(* Logix 5000 project; controller cal1632 1756-L62 rev 16.20; software revision 16.05 *)

TASK MainTask (continuous, watchdog 500 ms) : P01_System, P02_MOP_HMI_Iface, P11_Zone_1, P12_Zone_2, P13_Zone_3, P19_Advanced_Cooling, P20_Letoff, P21_Splice_Press, P22_Tension_Stand_1

MODULES
   Local : 1756-L62 (ICP 0, rev 16.20)
      p00_di_01 : 1756-IB16 (ICP 4, rev 3.1, Input RPI 20 ms)
      p00_di_02 : 1756-IB16 (ICP 5, rev 3.1, Input RPI 20 ms)
      p00_di_03 : 1756-IB16 (ICP 6, rev 3.1, Input RPI 20 ms)
      p00_do_01 : 1756-OA16I (ICP 7, rev 3.1, Output RPI 20 ms)
      p00_ai_01 : 1756-IF16 (ICP 3, rev 1.1, Input RPI 100 ms)
      Enet_A : 1756-ENBT (Ethernet 10.0.0.1, ICP 1, rev 4.1)
         p00_io_letoff : 1794-AENT (Ethernet 10.0.0.10, rev 3.1, Output RPI 25 ms)
            p00_io_letoff_do_01 : vendor 1 type 7 code 35 (Flex 3, rev 1.1)
            p00_io_letoff_di_01 : 1794-IB16 (Flex 4, rev 1.1)
            p00_io_letoff_di_02 : 1794-IB16 (Flex 5, rev 1.1)
            p00_io_letoff_di_03 : 1794-IB16 (Flex 6, rev 1.1)
            p00_io_letoff_di_04 : 1794-IB16 (Flex 7, rev 1.1)
            p00_io_letoff_ao_01 : 1794-OE4 (Flex 0, rev 2.1, Output RPI 80 ms)
            p00_io_letoff_ai_01 : vendor 1 type 10 code 25 (Flex 1, rev 2.1, Input RPI 80 ms)
            p00_io_letoff_tc_01 : vendor 1 type 10 code 28 (Flex 2, rev 1.1, Input RPI 80 ms)
         p00_io_oven : 1794-AENT (Ethernet 10.0.0.11, rev 3.1, Output RPI 25 ms)
            p00_io_oven_di_01 : 1794-IB16 (Flex 3, rev 1.1)
            p00_io_oven_di_02 : 1794-IB16 (Flex 4, rev 1.1)
            p00_io_oven_di_03 : 1794-IB16 (Flex 5, rev 1.1)
            p00_io_oven_ai_01 : vendor 1 type 10 code 25 (Flex 1, rev 2.1, Input RPI 80 ms)
            p00_io_oven_tc_01 : vendor 1 type 10 code 28 (Flex 2, rev 1.1, Input RPI 80 ms)
            p00_io_oven_ao_01 : 1794-OE4 (Flex 0, rev 2.1, Output RPI 80 ms)
         p00_io_winder : 1794-AENT (Ethernet 10.0.0.12, rev 3.1, Output RPI 25 ms)
            p00_io_winder_di_01 : 1794-IB16 (Flex 5, rev 1.1)
            p00_io_winder_do_01 : vendor 1 type 7 code 35 (Flex 4, rev 1.1)
            p00_io_winder_di_02 : 1794-IB16 (Flex 6, rev 1.1)
            p00_io_winder_ao_02 : 1794-OE4 (Flex 1, rev 2.1, Output RPI 80 ms)
            p00_io_winder_ai_01 : vendor 1 type 10 code 25 (Flex 2, rev 2.1, Input RPI 80 ms)
            p00_io_winder_tc_01 : vendor 1 type 10 code 28 (Flex 3, rev 1.1, Input RPI 80 ms)
            p00_io_winder_ao_01 : 1794-OE4 (Flex 0, rev 2.1, Output RPI 80 ms)
         p00_io_line : 1794-AENT (Ethernet 10.0.0.13, rev 3.1, Output RPI 25 ms)
            p00_io_line_do_01 : vendor 1 type 7 code 35 (Flex 1, rev 1.1)
            p00_io_line_di_01 : 1794-IB16 (Flex 2, rev 1.1)
            p00_io_line_di_02 : 1794-IB16 (Flex 3, rev 1.1)
            p00_io_line_ao_01 : 1794-OE4 (Flex 0, rev 2.1, Output RPI 80 ms)
         p00_io_prc : 1794-AENT (Ethernet 10.0.0.14, rev 3.1, Output RPI 25 ms)
            p00_io_prc_di_01 : 1794-IB16 (Flex 1, rev 1.1)
            p00_io_prc_do_01 : vendor 1 type 7 code 35 (Flex 0, rev 1.1)
         p00_vfd_imp_supply : ETHERNET-MODULE (Ethernet 10.0.0.50, rev 1.1, Output RPI 50 ms)
         p00_vfd_z1_recirc : ETHERNET-MODULE (Ethernet 10.0.0.51, rev 1.1, Output RPI 50 ms)
         p00_vfd_z1_exhaust : ETHERNET-MODULE (Ethernet 10.0.0.52, rev 1.1, Output RPI 50 ms)
         p00_vfd_z2_recirc : ETHERNET-MODULE (Ethernet 10.0.0.53, rev 1.1, Output RPI 50 ms)
         p00_vfd_z2_exhaust : ETHERNET-MODULE (Ethernet 10.0.0.54, rev 1.1, Output RPI 50 ms)
         p00_vfd_z3_exhaust : ETHERNET-MODULE (Ethernet 10.0.0.56, rev 1.1, Output RPI 50 ms)
         p00_vfd_z3_recirc : ETHERNET-MODULE (Ethernet 10.0.0.55, rev 1.1, Output RPI 50 ms)
      Enet_B : 1756-ENBT (ICP 2, Ethernet 10.0.1.1, rev 4.1)
         p00_vfd_loa : ETHERNET-MODULE (Ethernet 10.0.1.10, rev 1.1, Output RPI 10 ms)
         p00_vfd_lob : ETHERNET-MODULE (Ethernet 10.0.1.11, rev 1.1, Output RPI 10 ms)
         p00_vfd_lo_turret : ETHERNET-MODULE (Ethernet 10.0.1.12, rev 1.1, Output RPI 10 ms)
         p00_vfd_ts1 : ETHERNET-MODULE (Ethernet 10.0.1.13, rev 1.1, Output RPI 10 ms)
         p00_vfd_mtr : ETHERNET-MODULE (Ethernet 10.0.1.14, rev 1.1, Output RPI 10 ms)
         p00_srv_mtr_os : ETHERNET-MODULE (Ethernet 10.0.1.15, rev 1.1, Output RPI 10 ms)
         p00_srv_mtr_ds : ETHERNET-MODULE (Ethernet 10.0.1.16, rev 1.1, Output RPI 10 ms)
         p00_vfd_ts2 : ETHERNET-MODULE (Ethernet 10.0.1.17, rev 1.1, Output RPI 10 ms)
         p00_vfd_slitter : ETHERNET-MODULE (Ethernet 10.0.1.18, rev 1.1, Output RPI 10 ms)
         p00_vfd_wdr_turret : ETHERNET-MODULE (Ethernet 10.0.1.19, rev 1.1, Output RPI 10 ms)
         p00_vfd_wda : ETHERNET-MODULE (Ethernet 10.0.1.20, rev 1.1, Output RPI 10 ms)
         p00_vfd_wdb : ETHERNET-MODULE (Ethernet 10.0.1.21, rev 1.1, Output RPI 10 ms)
         p00_vfd_sprng : ETHERNET-MODULE (Ethernet 10.0.1.22, rev 1.1, Output RPI 10 ms)
END_MODULES

TYPE Accumulator :
STRUCT
   OUT_Not_EStop : BOOL;   // E-Stop Not Requested
   OUT_Not_Fast_Stop : BOOL;   // Fast Stop Not Requested
   OUT_Not_Normal_Stop : BOOL;   // Normal Stop Not Requested
   OUT_Request_Line_Slowdown : BOOL;   // Request Line Slowdown
   OUT_Full : BOOL;   // Accumulator is Full
   OUT_Empty : BOOL;   // Accumulator is Empty
   OUT_Alarm : BOOL;   // Alarm Exists
   OUT_Unack_Alarm : BOOL;   // Unacknowledged Alarm Exists
   OUT_Warning : BOOL;   // Warning Exists
   OUT_Unack_Warning : BOOL;   // Unacknowledged Warning Exists
   OUT_control_limit : BOOL;   // Control Limit Position
   OUT_Speed : REAL;   // Output Speed
   OUT_Nip_Close : BOOL;   // Nip Close Request
   IN_Speed : REAL;   // Input Speed
   OUT_Acc_Payout : BOOL;   // Accumulator Payout
   OUT_Close_Nip : BOOL;   // Close Nip
   OUT_Acc_Fill_Request : BOOL;   // Accumulator Fill Request
END_STRUCT
END_TYPE

TYPE acs800_di_normal :
STRUCT
   faulted : BOOL;
   warning : BOOL;
   running_fwd : BOOL;
   running_rev : BOOL;
   ready : BOOL;
   ctrl_from_net : BOOL;
   ref_from_net : BOOL;
   at_reference : BOOL;
END_STRUCT
END_TYPE

TYPE acs800_do_normal :
STRUCT
   forward : BOOL;
   reverse : BOOL;
   fault_reset : BOOL;
   net_control : BOOL;
   net_reference : BOOL;
END_STRUCT
END_TYPE

TYPE hmi_dint :
STRUCT
   hmi : DINT[16];
   global : DINT[16];
   zone_1 : DINT[16];
   zone_2 : DINT[16];
   zone_3 : DINT[16];
   letoff : DINT[16];
   ts1 : DINT[16];
   ts2 : DINT[16];
   upl : DINT[16];
   lpl : DINT[16];
   wdr : DINT[16];
   wdt : DINT[16];
   splice : DINT[16];
   mrc : DINT[16];
   static : DINT[16];
   imp : DINT[16];
   misc : DINT[16];
   edg : DINT[16];
   slt : DINT[16];
   impreg : DINT[16];
   adv_cooling : DINT[16];
   retraction : DINT[16];
END_STRUCT
END_TYPE

TYPE hmi_real :
STRUCT
   hmi : REAL[112];
   global : REAL[112];
   zone_1 : REAL[112];
   zone_2 : REAL[112];
   zone_3 : REAL[112];
   letoff : REAL[112];
   ts1 : REAL[112];
   ts2 : REAL[112];
   upl : REAL[112];
   lpl : REAL[112];
   wdr : REAL[112];
   wdt : REAL[112];
   splice : REAL[112];
   mrc : REAL[112];
   static : REAL[112];
   impreg : REAL[112];
   misc : REAL[112];
   edg : REAL[112];
   slt : REAL[112];
   adv_cooling : REAL[112];
END_STRUCT
END_TYPE

TYPE recipe :
STRUCT
   name : STRING;
   comments : STRING;
   master_line_speed : REAL;
   zone_1 : zone;
   zone_2 : zone;
   zone_3 : zone;
   line_speed_sp : REAL;
   letoff_tension_sp : REAL;
   acc_tension_sp : REAL;
   acc_fill_pressure_sp : REAL;
   acc_counter_pressure_sp : REAL;
   cure_time_sp : REAL;
   platen_temp_sp : REAL;
   impreg_gap_sp : REAL;
   impreg_gap_ds_offset_sp : REAL;
   impreg_gap_os_offset_sp : REAL;
   impreg_supply_speed_sp : REAL;
   impreg_roll_speed_sp : REAL;
   ts1_mode_sp : REAL;
   ts1_tension_sp : REAL;
   ts1_stretch_sp : REAL;
   liner_winder_brake_sp : REAL;
   slitter_speed_sp : REAL;
   adv_cooling_temp_sp : REAL;
   ts2_tension_sp : REAL;
   lower_poly_tension_sp : REAL;
   lower_poly_b_tension_sp : REAL;
   upper_poly_tension_sp : REAL;
   upper_poly_b_tension_sp : REAL;
   winder_tension_sp : REAL;
   winder_mode_sp : REAL;
   winder_torque_sp : REAL;
   tension_deviation_sp : REAL;
END_STRUCT
END_TYPE

TYPE routine :
STRUCT
   comment : DINT;
   oneshot : DINT;
   fault : DINT;
   fault_ack : DINT;
   fault1 : DINT;
   fault1_ack : DINT;
   warning : DINT;
   warning_ack : DINT;
   unack_fault : BOOL;
   unack_warning : BOOL;
   state : DINT;
END_STRUCT
END_TYPE

TYPE servo_di :
STRUCT
   mode_bit_0 : BOOL;
   mode_bit_1 : BOOL;
   homed : BOOL;
   stand_still : BOOL;
   at_target_pos : BOOL;
   command_change : BOOL;
   operator_mode_error : BOOL;
   drive_does_not_follow : BOOL;
   actual_op_mode_bit_0 : BOOL;
   actual_op_mode_bit_1 : BOOL;
   class_3_diagnostic : BOOL;
   class_2_diagnostic : BOOL;
   class_1_diagnostic : BOOL;
   operation_bit_14 : BOOL;
   operation_bit_15 : BOOL;
END_STRUCT
END_TYPE

TYPE servo_do :
STRUCT
   command_value_accept : BOOL;
   fault_reset : BOOL;
   jog_forward : BOOL;
   jog_reverse : BOOL;
   jog_enable : BOOL;
   drive_halt_0_halt : BOOL;
   drive_enable : BOOL;
   ready_for_operation_bit_16 : BOOL;
   ready_for_operation_bit_17 : BOOL;
END_STRUCT
END_TYPE

TYPE Setpoint :   // ******************** DO NOT CHANGE ORDER OF TAGS ******************** ****
STRUCT
   SP : REAL;   // Setpoint
   Lo : REAL;   // Lo
   Hi : REAL;   // Hi
END_STRUCT
END_TYPE

TYPE vfd_data :
STRUCT
   In_OutputFreq : DINT;
   In_RPM : DINT;
   In_OutputCurrent : DINT;
   In_MaximumFreq : DINT;
   In_MotorNPHz : DINT;
   In_MotorNPRPM : DINT;
   In_DriveStatus : DINT;
   Out_CommandedFreq : DINT;
   Out_DriveLogicRslt : DINT;
   Out_CommandedRPM : DINT;
   In_DriveStatus_Ready : BOOL;
   In_DriveStatus_Active : BOOL;
   In_DriveStatus_Faulted : BOOL;
   In_DriveStatus_Net : BOOL;
   In_DriveStatus_AtReference : BOOL;
   Out_DriveLogicRslt_Stop : BOOL;
   Out_DriveLogicRslt_Start : BOOL;
   Out_DriveLogicRslt_ClearFault : BOOL;
   Out_DriveLogicRslt_Forward : BOOL;
   Out_DriveLogicRslt_Reverse : BOOL;
END_STRUCT
END_TYPE

TYPE zone :
STRUCT
   recirc_sp : REAL;
   exhaust_sp : REAL;
   temp_sp : REAL;
END_STRUCT
END_TYPE

ADD_ON_INSTRUCTION ABB_PROTOCOL_VFD   (* revision 1.0 *)
VAR_INPUT
   STATUS_WORD : INT; {required}
END_VAR
VAR_OUTPUT
   CONTROL_WORD : INT; {required}
END_VAR
VAR_INPUT
   DRIVE_NOT_READY_FAULT : BOOL;
END_VAR
VAR_OUTPUT
   OUT_FAULT : BOOL; {visible}
   OUT_ALARM : BOOL; {visible}
   OUT_ENABLED : BOOL; {visible}
END_VAR
VAR_INPUT
   IN_START : BOOL; {required}
   IN_GLOBAL_RESET : BOOL; {required}
   IN_DRIVE_PERMISSIVE : BOOL; {required}
END_VAR
VAR
   run_permissive : BOOL;
   enable_drives : BOOL;
   request_run : BOOL;
   drive_on_request : BOOL;
   seq : routine;
   step_3_timer : TIMER := (PRE := 500);
   fault_timer : TIMER := (PRE := 2000);
END_VAR

ROUTINE Logic   (* ladder *)
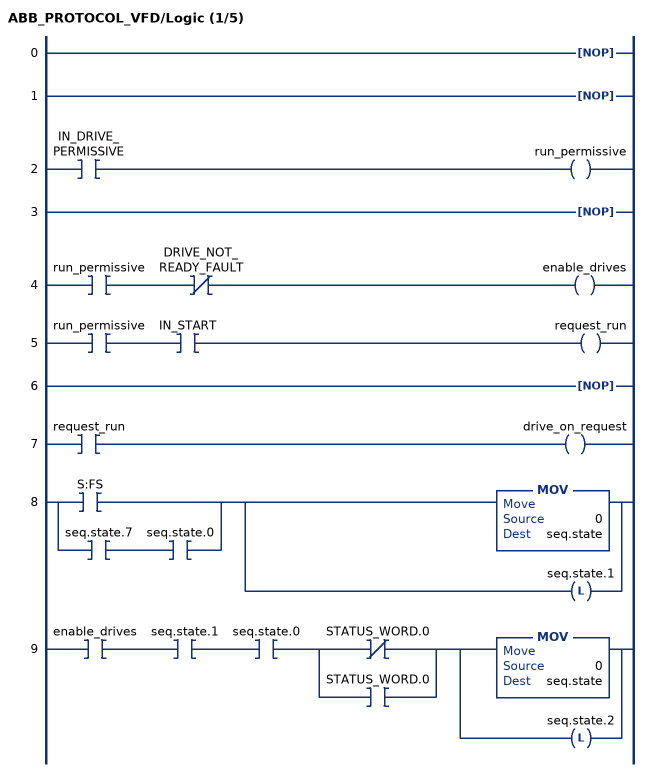
   0: NOP();
   1: NOP();
   2: XIC(IN_DRIVE_PERMISSIVE)OTE(run_permissive);
   3: NOP();
   4: XIC(run_permissive)XIO(DRIVE_NOT_READY_FAULT)OTE(enable_drives);
   5: XIC(run_permissive)XIC(IN_START)OTE(request_run);
   6: NOP();
   7: XIC(request_run)OTE(drive_on_request);
   8: [XIC(S:FS) ,XIC(seq.state.7) XIC(seq.state.0) ][MOV(0,seq.state) ,OTL(seq.state.1) ];
   9: XIC(enable_drives)XIC(seq.state.1)XIC(seq.state.0)[XIO(STATUS_WORD.0) ,XIC(STATUS_WORD.0) ][MOV(0,seq.state) ,OTL(seq.state.2) ];
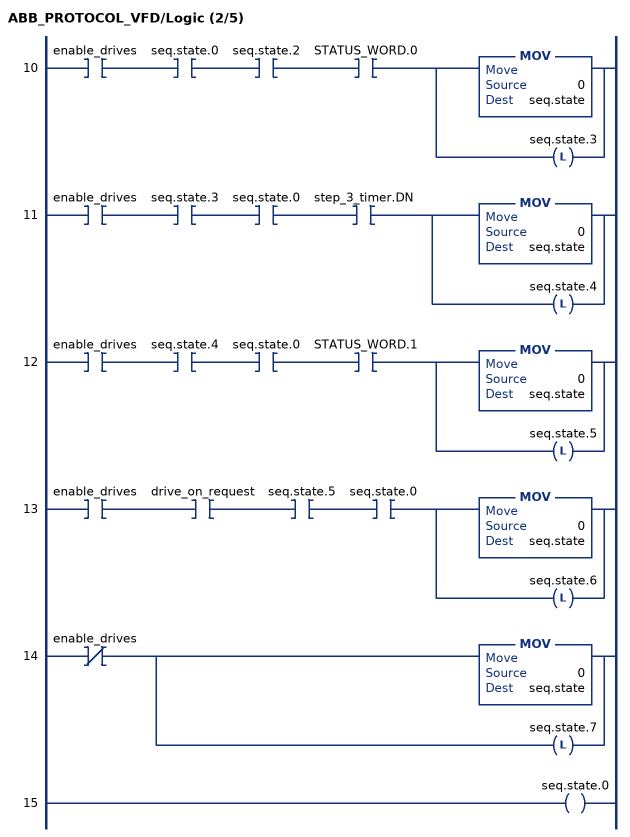
   10: XIC(enable_drives)XIC(seq.state.0)XIC(seq.state.2)XIC(STATUS_WORD.0)[MOV(0,seq.state) ,OTL(seq.state.3) ];
   11: XIC(enable_drives)XIC(seq.state.3)XIC(seq.state.0)XIC(step_3_timer.DN)[MOV(0,seq.state) ,OTL(seq.state.4) ];
   12: XIC(enable_drives)XIC(seq.state.4)XIC(seq.state.0)XIC(STATUS_WORD.1)[MOV(0,seq.state) ,OTL(seq.state.5) ];
   13: XIC(enable_drives)XIC(drive_on_request)XIC(seq.state.5)XIC(seq.state.0)[MOV(0,seq.state) ,OTL(seq.state.6) ];
   14: XIO(enable_drives)[MOV(0,seq.state) ,OTL(seq.state.7) ];
   15: OTE(seq.state.0);
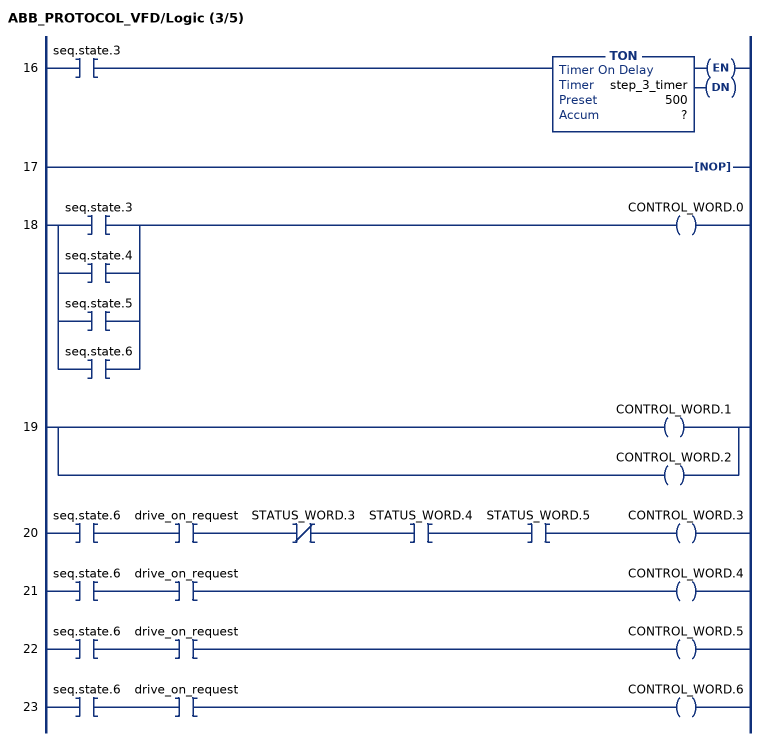
   16: XIC(seq.state.3)TON(step_3_timer,?,?);
   17: NOP();
   18: [XIC(seq.state.3) ,XIC(seq.state.4) ,XIC(seq.state.5) ,XIC(seq.state.6) ]OTE(CONTROL_WORD.0);
   19: [OTE(CONTROL_WORD.1) ,OTE(CONTROL_WORD.2) ];
   20: XIC(seq.state.6)XIC(drive_on_request)XIO(STATUS_WORD.3)XIC(STATUS_WORD.4)XIC(STATUS_WORD.5)OTE(CONTROL_WORD.3);
   21: XIC(seq.state.6)XIC(drive_on_request)OTE(CONTROL_WORD.4);
   22: XIC(seq.state.6)XIC(drive_on_request)OTE(CONTROL_WORD.5);
   23: XIC(seq.state.6)XIC(drive_on_request)OTE(CONTROL_WORD.6);
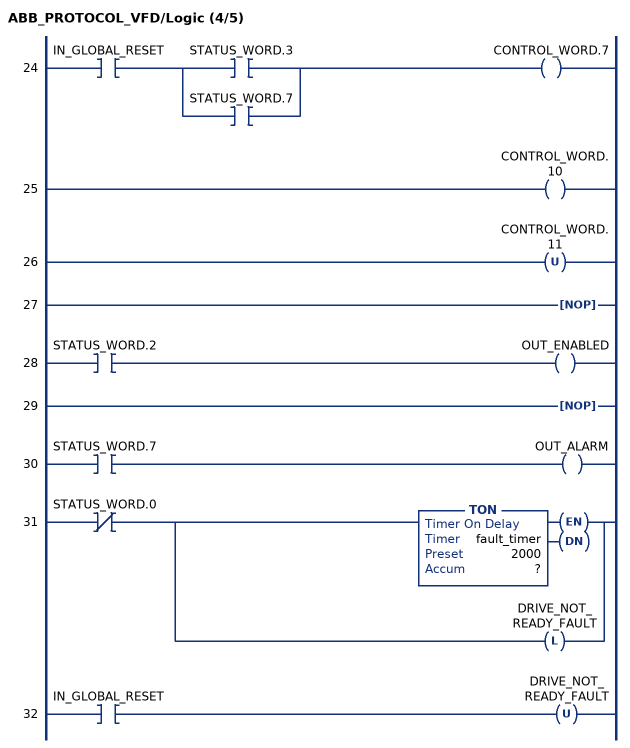
   24: XIC(IN_GLOBAL_RESET)[XIC(STATUS_WORD.3) ,XIC(STATUS_WORD.7) ]OTE(CONTROL_WORD.7);
   25: OTE(CONTROL_WORD.10);
   26: OTU(CONTROL_WORD.11);
   27: NOP();
   28: XIC(STATUS_WORD.2)OTE(OUT_ENABLED);
   29: NOP();
   30: XIC(STATUS_WORD.7)OTE(OUT_ALARM);
   31: XIO(STATUS_WORD.0)[TON(fault_timer,?,?) ,OTL(DRIVE_NOT_READY_FAULT) ];
   32: XIC(IN_GLOBAL_RESET)OTU(DRIVE_NOT_READY_FAULT);
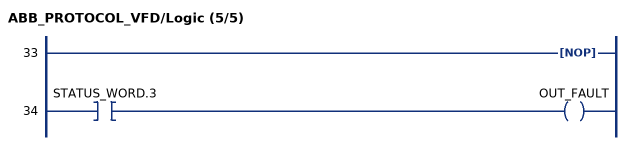
   33: NOP();
   34: XIC(STATUS_WORD.3)OTE(OUT_FAULT);
END_ROUTINE
END_ADD_ON_INSTRUCTION

ADD_ON_INSTRUCTION ARM_PID   (* revision 1.0 *)
VAR_IN_OUT
   PID : PID; {required}
END_VAR
VAR_INPUT
   NOBC : BOOL; {required}
   CA : BOOL; {required}
   Min : REAL; {required}
   Max : REAL; {required}
END_VAR

ROUTINE Logic   (* ladder *)
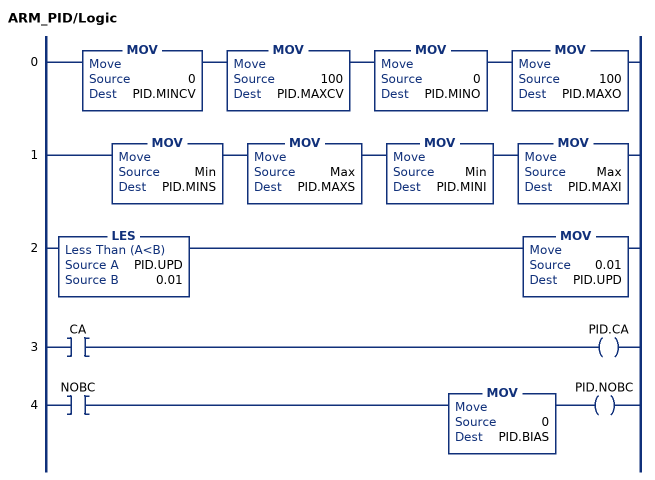
   0: MOV(0,PID.MINCV)MOV(100,PID.MAXCV)MOV(0,PID.MINO)MOV(100,PID.MAXO);
   1: MOV(Min,PID.MINS)MOV(Max,PID.MAXS)MOV(Min,PID.MINI)MOV(Max,PID.MAXI);
   2: LES(PID.UPD,0.01)MOV(0.01,PID.UPD);
   3: XIC(CA)OTE(PID.CA);
   4: XIC(NOBC)MOV(0,PID.BIAS)OTE(PID.NOBC);
END_ROUTINE
END_ADD_ON_INSTRUCTION

ADD_ON_INSTRUCTION Limit_Clamp   (* revision 1.0 *)
VAR_INPUT
   max : REAL; {required}
END_VAR
VAR_IN_OUT
   variable : REAL; {required}
END_VAR
VAR_INPUT
   min : REAL; {required}
END_VAR

ROUTINE Logic   (* ladder *)
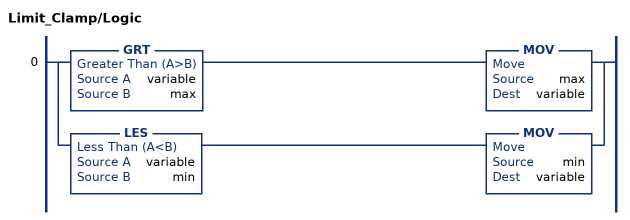
   0: [GRT(variable,max) MOV(max,variable) ,LES(variable,min) MOV(min,variable) ];
END_ROUTINE
END_ADD_ON_INSTRUCTION

ADD_ON_INSTRUCTION Ramp_Test   (* revision 1.0 *)
VAR_INPUT
   SP : REAL; {required}
   Rate : REAL; {required}
   ScanTime : REAL; {required}
END_VAR
VAR_IN_OUT
   PV : REAL; {required}
END_VAR
VAR
   request_decel : BOOL;
   request_accel : BOOL;
END_VAR

ROUTINE Logic   (* ladder *)
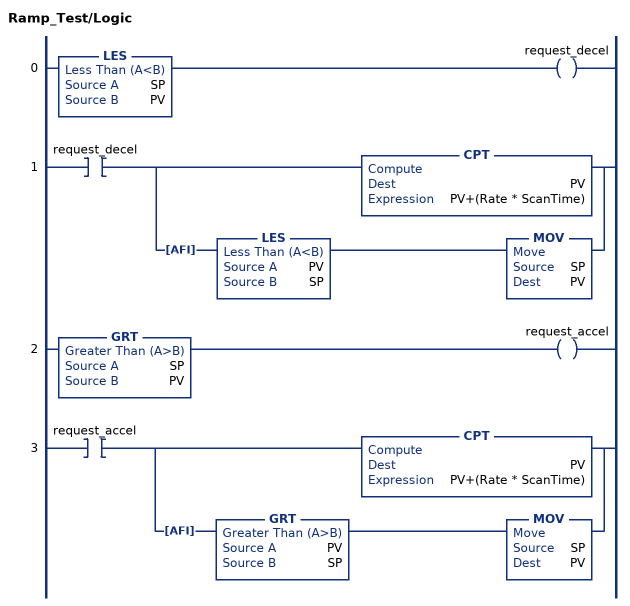
   0: LES(SP,PV)OTE(request_decel);
   1: XIC(request_decel)[CPT(PV,PV+(Rate * ScanTime)) ,AFI() LES(PV,SP) MOV(SP,PV) ];
   2: GRT(SP,PV)OTE(request_accel);
   3: XIC(request_accel)[CPT(PV,PV+(Rate * ScanTime)) ,AFI() GRT(PV,SP) MOV(SP,PV) ];
END_ROUTINE
END_ADD_ON_INSTRUCTION

ADD_ON_INSTRUCTION SYS_ACC_DEC_RAMP   (* revision 1.0 *)
VAR_INPUT
   IN_selected_line_speed : REAL; {required}
   IN_param_master_accel_rate : REAL; {required}
   IN_param_master_decel_rate : REAL; {required}
   IN_last_scan_s : REAL; {required}
END_VAR
VAR_IN_OUT
   IN_OUT_master_ramped_speed : REAL; {required}
END_VAR
VAR
   p01r03_last_scan_ms : DINT;
   local_last_scan_ms : DINT;
END_VAR

ROUTINE Logic   (* ladder *)
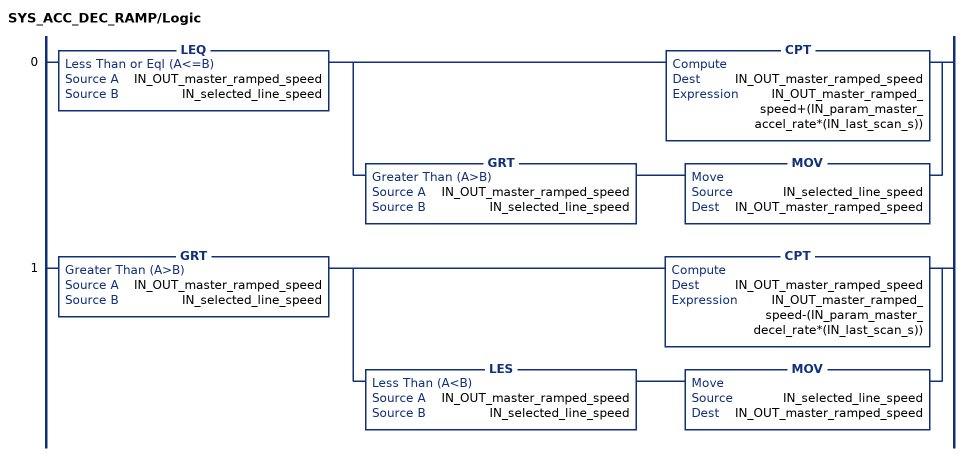
   0: LEQ(IN_OUT_master_ramped_speed,IN_selected_line_speed)[CPT(IN_OUT_master_ramped_speed,IN_OUT_master_ramped_speed+(IN_param_master_accel_rate*(IN_last_scan_s))) ,GRT(IN_OUT_master_ramped_speed,IN_selected_line_speed) MOV(IN_selected_line_speed,IN_OUT_master_ramped_speed) ];
   1: GRT(IN_OUT_master_ramped_speed,IN_selected_line_speed)[CPT(IN_OUT_master_ramped_speed,IN_OUT_master_ramped_speed-(IN_param_master_decel_rate*(IN_last_scan_s))) ,LES(IN_OUT_master_ramped_speed,IN_selected_line_speed) MOV(IN_selected_line_speed,IN_OUT_master_ramped_speed) ];
END_ROUTINE
END_ADD_ON_INSTRUCTION

ADD_ON_INSTRUCTION sys_Acknowledge   (* revision 1.0 *)
VAR_INPUT
   EnableIn1 : BOOL;   // Enable Input - System Defined Parameter
END_VAR
VAR_OUTPUT
   EnableOut1 : BOOL;   // Enable Output - System Defined Parameter
END_VAR
VAR_IN_OUT
   Ack : DINT; {required}
END_VAR
VAR_INPUT
   Alarm : DINT; {required}
END_VAR

ROUTINE Logic   (* ladder *)
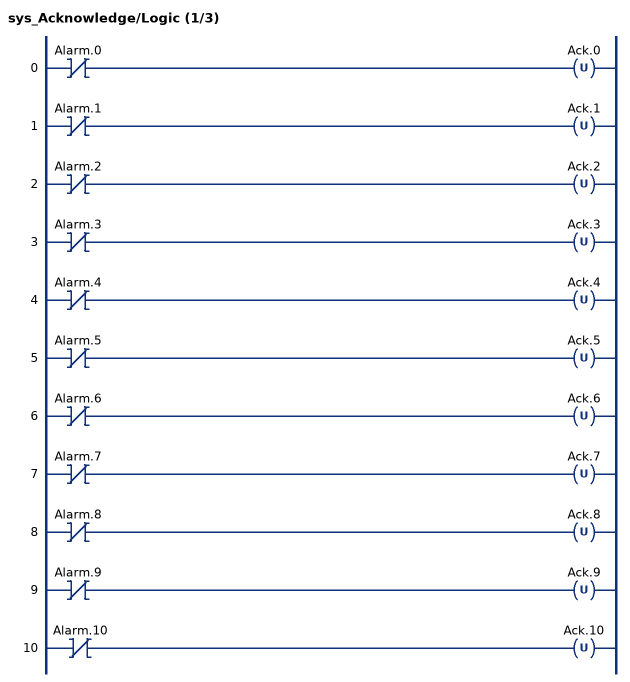
   0: XIO(Alarm.0)OTU(Ack.0);
   1: XIO(Alarm.1)OTU(Ack.1);
   2: XIO(Alarm.2)OTU(Ack.2);
   3: XIO(Alarm.3)OTU(Ack.3);
   4: XIO(Alarm.4)OTU(Ack.4);
   5: XIO(Alarm.5)OTU(Ack.5);
   6: XIO(Alarm.6)OTU(Ack.6);
   7: XIO(Alarm.7)OTU(Ack.7);
   8: XIO(Alarm.8)OTU(Ack.8);
   9: XIO(Alarm.9)OTU(Ack.9);
   10: XIO(Alarm.10)OTU(Ack.10);
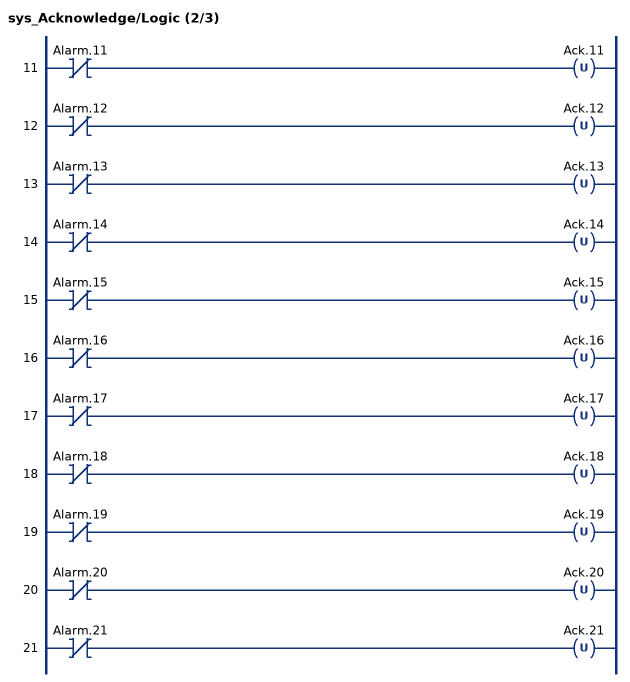
   11: XIO(Alarm.11)OTU(Ack.11);
   12: XIO(Alarm.12)OTU(Ack.12);
   13: XIO(Alarm.13)OTU(Ack.13);
   14: XIO(Alarm.14)OTU(Ack.14);
   15: XIO(Alarm.15)OTU(Ack.15);
   16: XIO(Alarm.16)OTU(Ack.16);
   17: XIO(Alarm.17)OTU(Ack.17);
   18: XIO(Alarm.18)OTU(Ack.18);
   19: XIO(Alarm.19)OTU(Ack.19);
   20: XIO(Alarm.20)OTU(Ack.20);
   21: XIO(Alarm.21)OTU(Ack.21);
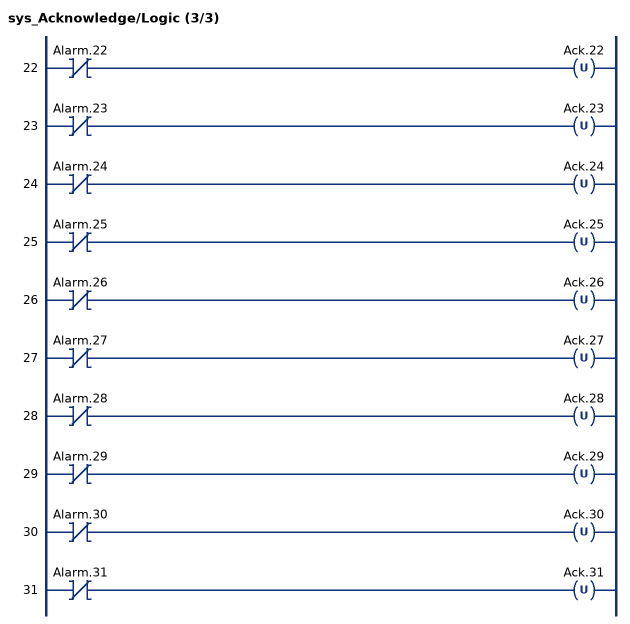
   22: XIO(Alarm.22)OTU(Ack.22);
   23: XIO(Alarm.23)OTU(Ack.23);
   24: XIO(Alarm.24)OTU(Ack.24);
   25: XIO(Alarm.25)OTU(Ack.25);
   26: XIO(Alarm.26)OTU(Ack.26);
   27: XIO(Alarm.27)OTU(Ack.27);
   28: XIO(Alarm.28)OTU(Ack.28);
   29: XIO(Alarm.29)OTU(Ack.29);
   30: XIO(Alarm.30)OTU(Ack.30);
   31: XIO(Alarm.31)OTU(Ack.31);
END_ROUTINE
END_ADD_ON_INSTRUCTION

ADD_ON_INSTRUCTION SYS_ENC   (* revision 1.0 *)
VAR_INPUT
   IN_State : DINT; {required}
END_VAR
VAR_OUTPUT
   OUT_Status : DINT; {required}
END_VAR

ROUTINE Logic   (* ladder *)
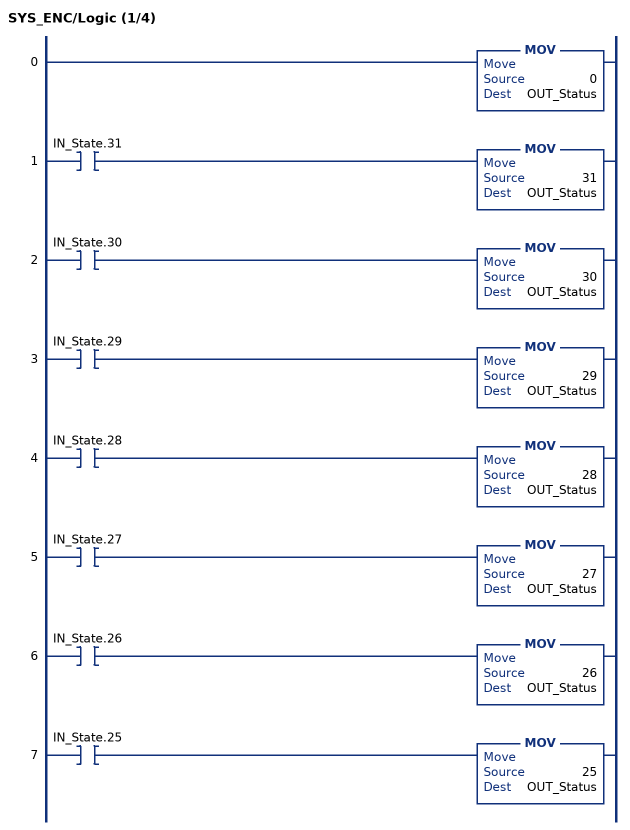
   0: MOV(0,OUT_Status);
   1: XIC(IN_State.31)MOV(31,OUT_Status);
   2: XIC(IN_State.30)MOV(30,OUT_Status);
   3: XIC(IN_State.29)MOV(29,OUT_Status);
   4: XIC(IN_State.28)MOV(28,OUT_Status);
   5: XIC(IN_State.27)MOV(27,OUT_Status);
   6: XIC(IN_State.26)MOV(26,OUT_Status);
   7: XIC(IN_State.25)MOV(25,OUT_Status);
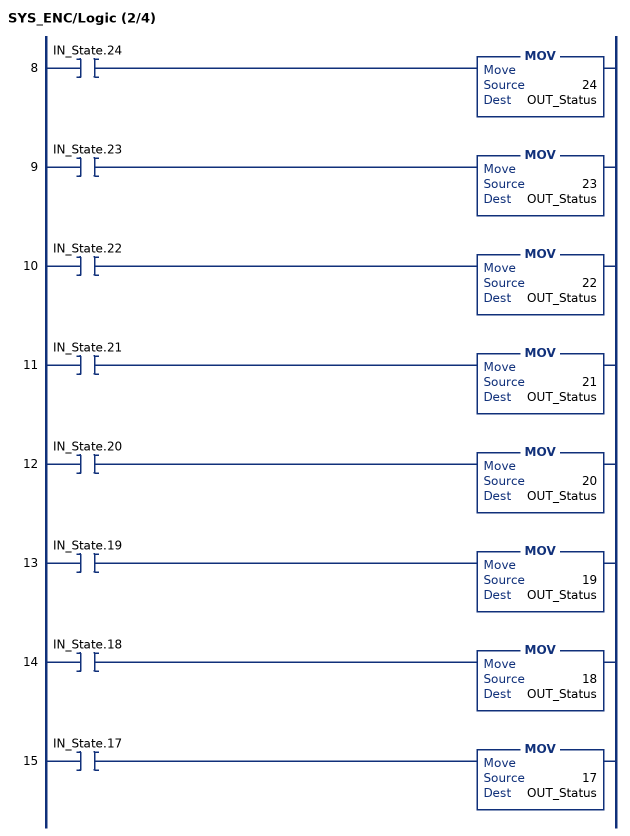
   8: XIC(IN_State.24)MOV(24,OUT_Status);
   9: XIC(IN_State.23)MOV(23,OUT_Status);
   10: XIC(IN_State.22)MOV(22,OUT_Status);
   11: XIC(IN_State.21)MOV(21,OUT_Status);
   12: XIC(IN_State.20)MOV(20,OUT_Status);
   13: XIC(IN_State.19)MOV(19,OUT_Status);
   14: XIC(IN_State.18)MOV(18,OUT_Status);
   15: XIC(IN_State.17)MOV(17,OUT_Status);
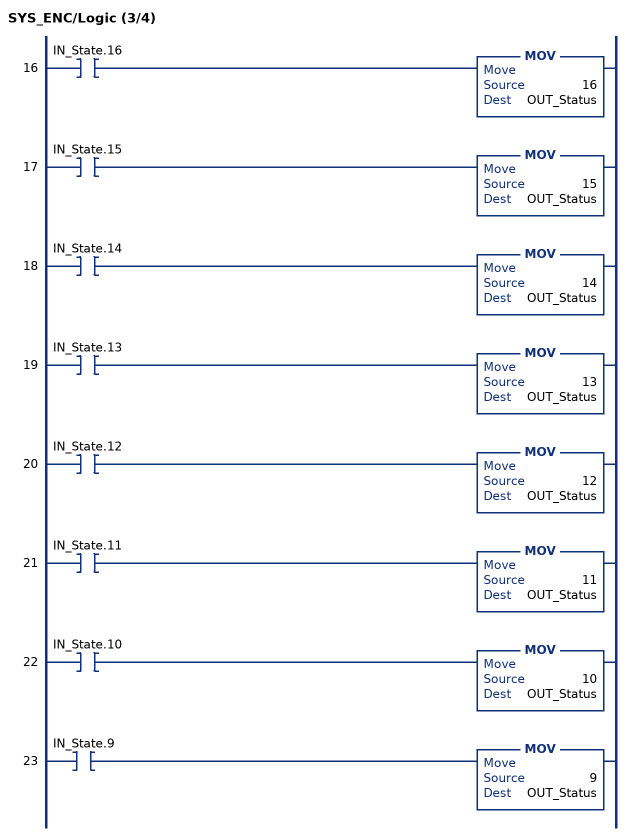
   16: XIC(IN_State.16)MOV(16,OUT_Status);
   17: XIC(IN_State.15)MOV(15,OUT_Status);
   18: XIC(IN_State.14)MOV(14,OUT_Status);
   19: XIC(IN_State.13)MOV(13,OUT_Status);
   20: XIC(IN_State.12)MOV(12,OUT_Status);
   21: XIC(IN_State.11)MOV(11,OUT_Status);
   22: XIC(IN_State.10)MOV(10,OUT_Status);
   23: XIC(IN_State.9)MOV(9,OUT_Status);
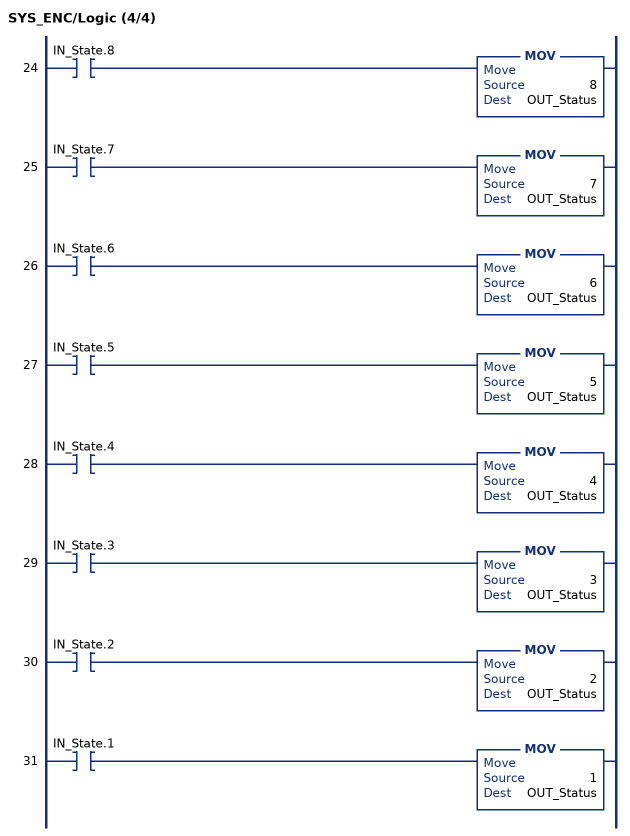
   24: XIC(IN_State.8)MOV(8,OUT_Status);
   25: XIC(IN_State.7)MOV(7,OUT_Status);
   26: XIC(IN_State.6)MOV(6,OUT_Status);
   27: XIC(IN_State.5)MOV(5,OUT_Status);
   28: XIC(IN_State.4)MOV(4,OUT_Status);
   29: XIC(IN_State.3)MOV(3,OUT_Status);
   30: XIC(IN_State.2)MOV(2,OUT_Status);
   31: XIC(IN_State.1)MOV(1,OUT_Status);
END_ROUTINE
END_ADD_ON_INSTRUCTION

ADD_ON_INSTRUCTION SYS_ENC_WITH_ZERO_BIT   (* revision 1.0 *)
VAR_INPUT
   IN_State : DINT; {required}
END_VAR
VAR_OUTPUT
   OUT_Status : DINT; {required}
END_VAR

ROUTINE Logic   (* ladder *)
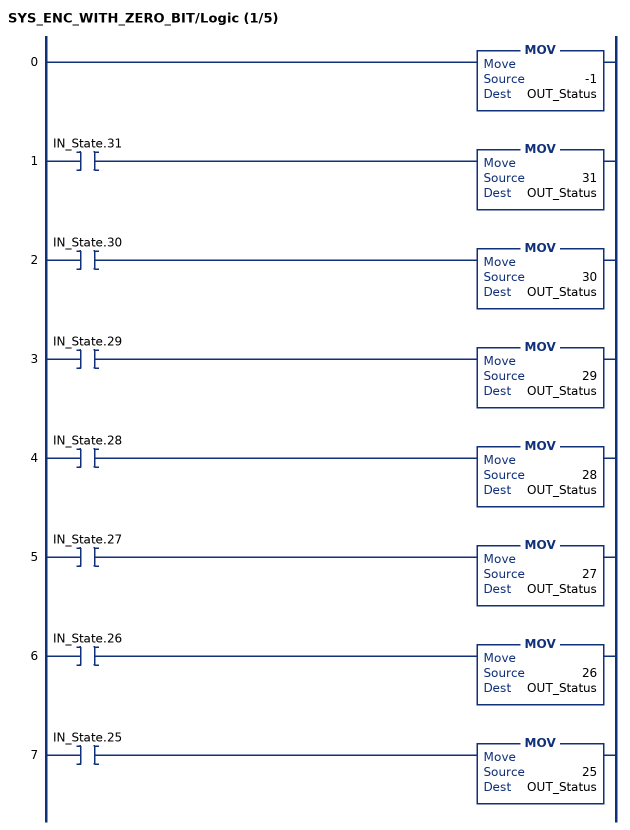
   0: MOV(-1,OUT_Status);
   1: XIC(IN_State.31)MOV(31,OUT_Status);
   2: XIC(IN_State.30)MOV(30,OUT_Status);
   3: XIC(IN_State.29)MOV(29,OUT_Status);
   4: XIC(IN_State.28)MOV(28,OUT_Status);
   5: XIC(IN_State.27)MOV(27,OUT_Status);
   6: XIC(IN_State.26)MOV(26,OUT_Status);
   7: XIC(IN_State.25)MOV(25,OUT_Status);
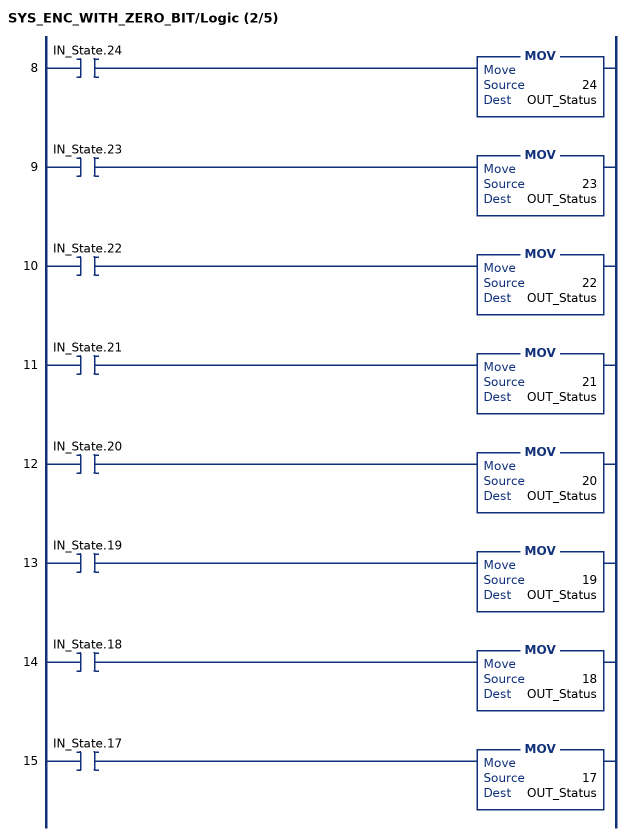
   8: XIC(IN_State.24)MOV(24,OUT_Status);
   9: XIC(IN_State.23)MOV(23,OUT_Status);
   10: XIC(IN_State.22)MOV(22,OUT_Status);
   11: XIC(IN_State.21)MOV(21,OUT_Status);
   12: XIC(IN_State.20)MOV(20,OUT_Status);
   13: XIC(IN_State.19)MOV(19,OUT_Status);
   14: XIC(IN_State.18)MOV(18,OUT_Status);
   15: XIC(IN_State.17)MOV(17,OUT_Status);
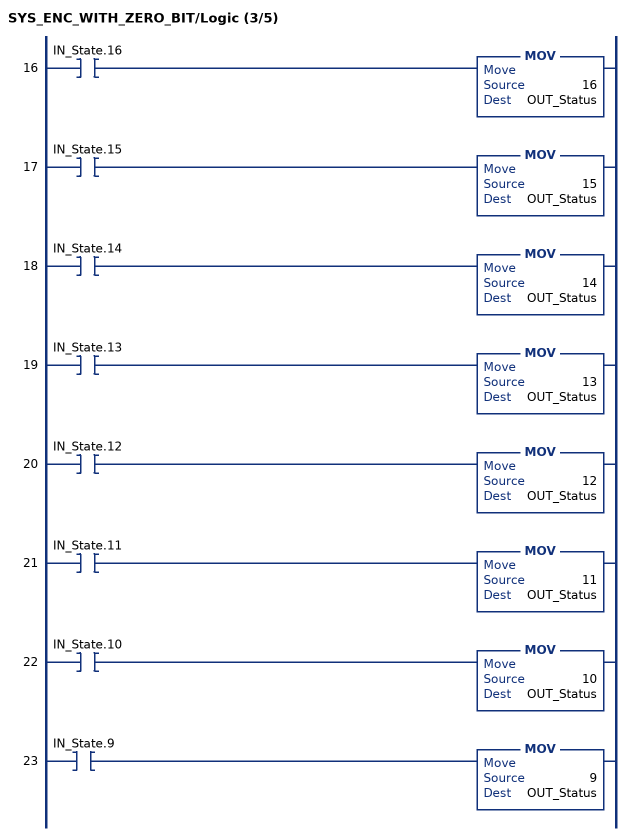
   16: XIC(IN_State.16)MOV(16,OUT_Status);
   17: XIC(IN_State.15)MOV(15,OUT_Status);
   18: XIC(IN_State.14)MOV(14,OUT_Status);
   19: XIC(IN_State.13)MOV(13,OUT_Status);
   20: XIC(IN_State.12)MOV(12,OUT_Status);
   21: XIC(IN_State.11)MOV(11,OUT_Status);
   22: XIC(IN_State.10)MOV(10,OUT_Status);
   23: XIC(IN_State.9)MOV(9,OUT_Status);
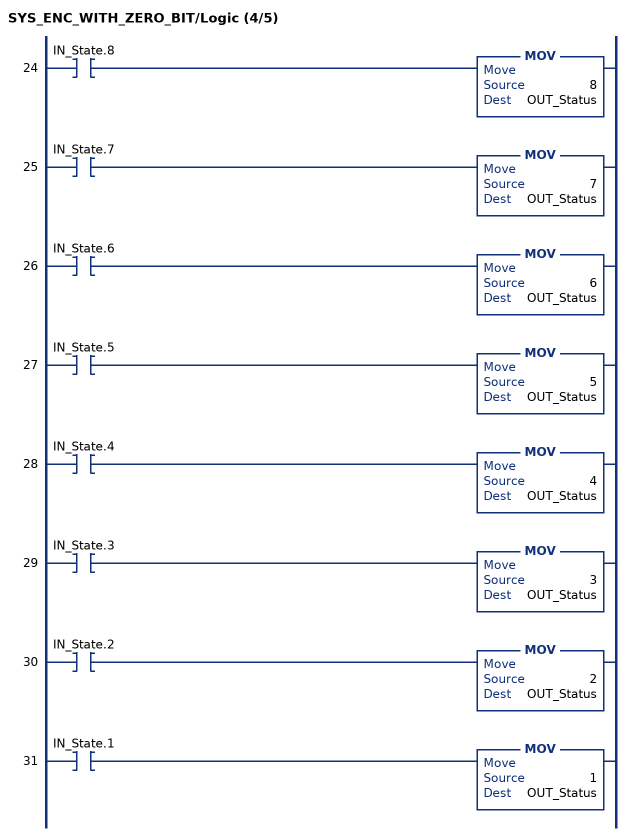
   24: XIC(IN_State.8)MOV(8,OUT_Status);
   25: XIC(IN_State.7)MOV(7,OUT_Status);
   26: XIC(IN_State.6)MOV(6,OUT_Status);
   27: XIC(IN_State.5)MOV(5,OUT_Status);
   28: XIC(IN_State.4)MOV(4,OUT_Status);
   29: XIC(IN_State.3)MOV(3,OUT_Status);
   30: XIC(IN_State.2)MOV(2,OUT_Status);
   31: XIC(IN_State.1)MOV(1,OUT_Status);
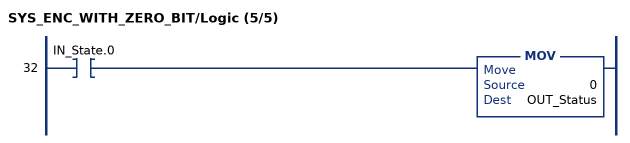
   32: XIC(IN_State.0)MOV(0,OUT_Status);
END_ROUTINE
END_ADD_ON_INSTRUCTION
